FUNCTION_BLOCK FB_TestObject EXTENDS FB_Object
VAR_INPUT
END_VAR
VAR_OUTPUT
END_VAR
VAR
    _nTest: INT;
END_VAR

PROPERTY nTest : INT
GET
nTest := THIS^._nTest;
END_GET
SET
THIS^._nTest := nTest;
END_SET
END_PROPERTY

END_FUNCTION_BLOCK

(* stored: Version 1.1.0.1, ProductVersion 3.1.4024.12
   POU FB_TestObject: Id {578513b7-8eb5-4b09-9ef8-d1a89742a507}, SpecialFunc None
   Property nTest: Id {a6ad0285-11ba-4447-8e13-ec96833e2cfc}
   Get Get: Id {8d4a4ec0-c987-40c5-90fa-89d52487441e}
   Set Set: Id {ffa5d75b-9dc8-4f5b-8520-f4eabd3d5234} *)
